SYSTEM Demo
  (* Version 1.0, 2020-01-11, Duc Do Tran *)
  APPLICATION SystemWithoutContract
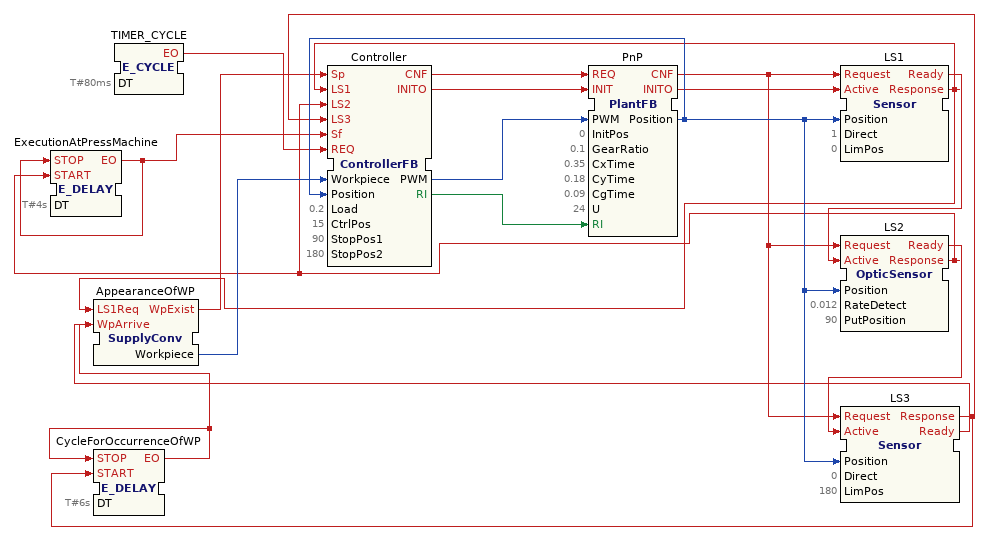
    FBS
      LS2 : OpticSensor(RateDetect := 0.012, PutPosition := 90);
      PnP : PlantFB(InitPos := 0, GearRatio := 0.1, CxTime := 0.35, CyTime := 0.18, CgTime := 0.09, U := 24);
      LS1 : Sensor(Direct := 1, LimPos := 0);
      LS3 : Sensor(Direct := 0, LimPos := 180);
      Controller : ControllerFB(Load := 0.2, CtrlPos := 15, StopPos1 := 90, StopPos2 := 180);
      AppearanceOfWP : SupplyConv;
      ExecutionAtPressMachine : E_DELAY(DT := T#4s);
      CycleForOccurrenceOfWP : E_DELAY(DT := T#6s);
      TIMER_CYCLE : E_CYCLE(DT := T#80ms);
    END_FBS
    EVENT_CONNECTIONS
      PnP.CNF TO LS1.Request;
      PnP.CNF TO LS2.Request;
      PnP.CNF TO LS3.Request;
      PnP.INITO TO LS1.Active;
      LS1.Ready TO LS2.Active;
      LS2.Ready TO LS3.Active;
      Controller.CNF TO PnP.REQ;
      Controller.INITO TO PnP.INIT;
      AppearanceOfWP.WpExist TO Controller.Sp;
      LS1.Response TO AppearanceOfWP.LS1Req;
      LS1.Response TO Controller.LS1;
      LS2.Response TO Controller.LS2;
      LS3.Response TO Controller.LS3;
      ExecutionAtPressMachine.EO TO Controller.Sf;
      ExecutionAtPressMachine.EO TO ExecutionAtPressMachine.STOP;
      CycleForOccurrenceOfWP.EO TO AppearanceOfWP.WpArrive;
      CycleForOccurrenceOfWP.EO TO CycleForOccurrenceOfWP.STOP;
      LS3.Response TO CycleForOccurrenceOfWP.START;
      LS3.Ready TO AppearanceOfWP.WpArrive;
      LS2.Response TO ExecutionAtPressMachine.START;
      TIMER_CYCLE.EO TO Controller.REQ;
    END_CONNECTIONS
    DATA_CONNECTIONS
      PnP.Position TO LS3.Position;
      PnP.Position TO LS2.Position;
      PnP.Position TO LS1.Position;
      Controller.PWM TO PnP.PWM;
      AppearanceOfWP.Workpiece TO Controller.Workpiece;
      PnP.Position TO Controller.Position;
    END_CONNECTIONS
    ADAPTER_CONNECTIONS
      Controller.RI TO PnP.RI;
    END_CONNECTIONS
  END_APPLICATION
  APPLICATION SystemApplyTimingContracts
    FBS
      LS2 : OpticSensor(RateDetect := 0.012, PutPosition := 90);
      ExecutionAtPressMachine : E_DELAY(DT := T#4000ms);
      SplitFirstOccurOfLS1 : SplitInitEv;
      TIMER_CYCLE : E_DELAY(DT := T#20ms);
      LS1ToLS2 : TCFB(QI := 1, GetTime := 0, SetTimeOut := 20.3, Specification := Reaction::q->e(i|=[3.5,4.8]s));
      LS2ToSf : TCFB(QI := 1, GetTime := 0, SetTimeOut := 20.3, Specification := Age::q->e(i|=[3.9,4.4]s));
      SfToLS3 : TCFB(QI := 1, GetTime := 0, SetTimeOut := 20.3, Specification := Reaction::q->e(i|=[4.1,4.6]s));
      LS3ToLS1 : TCFB(QI := 1, GetTime := 0, SetTimeOut := 20.3, Specification := Reaction::q->e(i|=[6.2,6.5]s));
      AppearanceOfWP : SupplyConv;
      PickAndPlaceRobot : PlantFB(InitPos := 0, GearRatio := 0.1, CxTime := 0.35, CyTime := 0.18, CgTime := 0.09, U := 24);
      CycleForOccurrenceOfWP : E_DELAY(DT := T#6000ms);
      LS1 : Sensor(Direct := 1, LimPos := 0);
      LS3 : Sensor(Direct := 0, LimPos := 180);
      Controller : ControllerFB(Load := 0.2, CtrlPos := 15, StopPos1 := 90, StopPos2 := 180);
      EnableCheck : EnableCheck(QIi := 1);
      OnOffLS1 : E_SWITCH(G := 1);
      OnOffLS2 : E_SWITCH(G := 1);
      OnOffLS3 : E_SWITCH(G := 1);
      OnOffFeedingSystem : E_SWITCH(G := 1);
      OnOffPressMachine : E_SWITCH(G := 1);
    END_FBS
    EVENT_CONNECTIONS
      LS2ToSf.Satisfied TO Controller.Sf;
      TIMER_CYCLE.EO TO TIMER_CYCLE.STOP;
      Controller.INITO TO PickAndPlaceRobot.INIT;
      LS2ToSf.INITO TO SfToLS3.INIT;
      SplitFirstOccurOfLS1.CNF TO AppearanceOfWP.LS1Req;
      EnableCheck.Satisfied TO Controller.LS1;
      ExecutionAtPressMachine.EO TO ExecutionAtPressMachine.STOP;
      LS2.Ready TO LS3.Active;
      SfToLS3.INITO TO LS3ToLS1.INIT;
      EnableCheck.Violated TO LS1ToLS2.ReqEvent;
      LS2ToSf.Satisfied TO SfToLS3.ReqEvent;
      CycleForOccurrenceOfWP.EO TO AppearanceOfWP.WpArrive;
      LS3ToLS1.CNF TO TIMER_CYCLE.START;
      EnableCheck.Satisfied TO LS1ToLS2.ReqEvent;
      LS2ToSf.CNF TO SfToLS3.REQ;
      SfToLS3.Satisfied TO Controller.LS3;
      LS2ToSf.Violated TO SfToLS3.ReqEvent;
      PickAndPlaceRobot.INITO TO TIMER_CYCLE.START;
      LS1ToLS2.Violated TO LS2ToSf.ReqEvent;
      SfToLS3.Violated TO LS3ToLS1.ReqEvent;
      TIMER_CYCLE.EO TO LS1ToLS2.REQ;
      LS3ToLS1.Violated TO EnableCheck.REQ;
      LS1ToLS2.Satisfied TO LS2ToSf.ReqEvent;
      LS3ToLS1.CNF TO Controller.REQ;
      LS1ToLS2.Satisfied TO Controller.LS2;
      LS3ToLS1.INITO TO LS1.Active;
      LS3.Response TO SfToLS3.RspEvent;
      LS1.Ready TO LS2.Active;
      LS3.Ready TO AppearanceOfWP.WpArrive;
      ExecutionAtPressMachine.EO TO LS2ToSf.RspEvent;
      LS1ToLS2.INITO TO LS2ToSf.INIT;
      SfToLS3.CNF TO LS3ToLS1.REQ;
      SplitFirstOccurOfLS1.NextTimes TO LS3ToLS1.RspEvent;
      AppearanceOfWP.WpExist TO Controller.Sp;
      LS3ToLS1.Satisfied TO EnableCheck.REQ;
      SfToLS3.Satisfied TO LS3ToLS1.ReqEvent;
      SplitFirstOccurOfLS1.FirstTime TO EnableCheck.REQ;
      LS2.Response TO LS1ToLS2.RspEvent;
      LS3ToLS1.INITO TO Controller.INIT;
      CycleForOccurrenceOfWP.EO TO CycleForOccurrenceOfWP.STOP;
      Controller.CNF TO PickAndPlaceRobot.REQ;
      LS1ToLS2.CNF TO LS2ToSf.REQ;
      LS1.Response TO SplitFirstOccurOfLS1.REQ;
      PickAndPlaceRobot.CNF TO OnOffLS3.EI;
      OnOffLS3.EO1 TO LS3.Request;
      PickAndPlaceRobot.CNF TO OnOffLS2.EI;
      OnOffLS2.EO1 TO LS2.Request;
      PickAndPlaceRobot.CNF TO OnOffLS1.EI;
      OnOffLS1.EO1 TO LS1.Request;
      LS3.Response TO OnOffFeedingSystem.EI;
      OnOffFeedingSystem.EO1 TO CycleForOccurrenceOfWP.START;
      LS1ToLS2.Satisfied TO OnOffPressMachine.EI;
      OnOffPressMachine.EO1 TO ExecutionAtPressMachine.START;
    END_CONNECTIONS
    DATA_CONNECTIONS
      PickAndPlaceRobot.Position TO LS3.Position;
      LS1ToLS2.QO TO LS2ToSf.QI;
      PickAndPlaceRobot.Position TO LS1.Position;
      Controller.PWM TO PickAndPlaceRobot.PWM;
      EnableCheck.OUT TO LS1ToLS2.QI;
      PickAndPlaceRobot.Position TO LS2.Position;
      LS2ToSf.QO TO SfToLS3.QI;
      PickAndPlaceRobot.Position TO Controller.Position;
      LS3ToLS1.QO TO EnableCheck.QIt;
      SfToLS3.QO TO LS3ToLS1.QI;
      AppearanceOfWP.Workpiece TO Controller.Workpiece;
    END_CONNECTIONS
    ADAPTER_CONNECTIONS
      Controller.RI TO PickAndPlaceRobot.RI;
    END_CONNECTIONS
  END_APPLICATION
  DEVICE FORTE_PC : FORTE_PC(MGR_ID := "localhost:61499")
    {SET_ATTRIBUTE(Profile, HOLOBLOC)} (* device profile *)
    RESOURCE CPU1 : EMB_RES
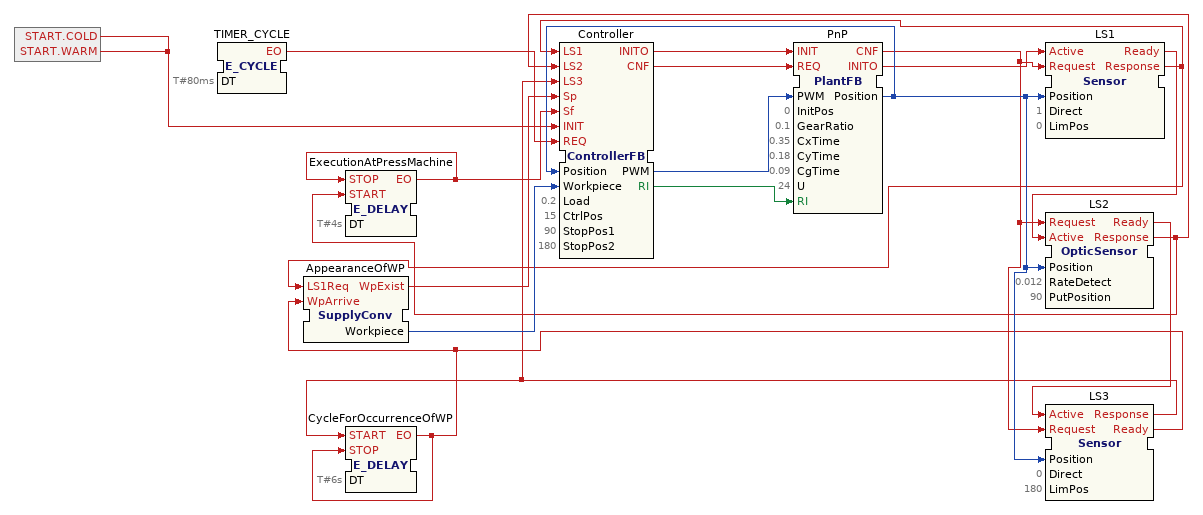
      FBS
        LS2 : OpticSensor(RateDetect := 0.012, PutPosition := 90);
        PnP : PlantFB(InitPos := 0, GearRatio := 0.1, CxTime := 0.35, CyTime := 0.18, CgTime := 0.09, U := 24);
        LS1 : Sensor(Direct := 1, LimPos := 0);
        LS3 : Sensor(Direct := 0, LimPos := 180);
        Controller : ControllerFB(Load := 0.2, CtrlPos := 15, StopPos1 := 90, StopPos2 := 180);
        AppearanceOfWP : SupplyConv;
        ExecutionAtPressMachine : E_DELAY(DT := T#4s);
        CycleForOccurrenceOfWP : E_DELAY(DT := T#6s);
        TIMER_CYCLE : E_CYCLE(DT := T#80ms);
      END_FBS
      EVENT_CONNECTIONS
        PnP.CNF TO LS2.Request;
        PnP.INITO TO LS1.Active;
        PnP.CNF TO LS1.Request;
        LS1.Ready TO LS2.Active;
        LS2.Ready TO LS3.Active;
        PnP.CNF TO LS3.Request;
        LS1.Response TO Controller.LS1;
        LS2.Response TO Controller.LS2;
        LS3.Response TO Controller.LS3;
        Controller.INITO TO PnP.INIT;
        Controller.CNF TO PnP.REQ;
        LS1.Response TO AppearanceOfWP.LS1Req;
        AppearanceOfWP.WpExist TO Controller.Sp;
        ExecutionAtPressMachine.EO TO ExecutionAtPressMachine.STOP;
        ExecutionAtPressMachine.EO TO Controller.Sf;
        LS3.Response TO CycleForOccurrenceOfWP.START;
        CycleForOccurrenceOfWP.EO TO CycleForOccurrenceOfWP.STOP;
        CycleForOccurrenceOfWP.EO TO AppearanceOfWP.WpArrive;
        LS3.Ready TO AppearanceOfWP.WpArrive;
        LS2.Response TO ExecutionAtPressMachine.START;
        START.COLD TO Controller.INIT;
        START.WARM TO Controller.INIT;
        TIMER_CYCLE.EO TO Controller.REQ;
      END_CONNECTIONS
      DATA_CONNECTIONS
        PnP.Position TO LS2.Position;
        PnP.Position TO LS1.Position;
        PnP.Position TO LS3.Position;
        PnP.Position TO Controller.Position;
        Controller.PWM TO PnP.PWM;
        AppearanceOfWP.Workpiece TO Controller.Workpiece;
      END_CONNECTIONS
      ADAPTER_CONNECTIONS
        Controller.RI TO PnP.RI;
      END_CONNECTIONS
    END_RESOURCE
    RESOURCE CPU2 : EMB_RES
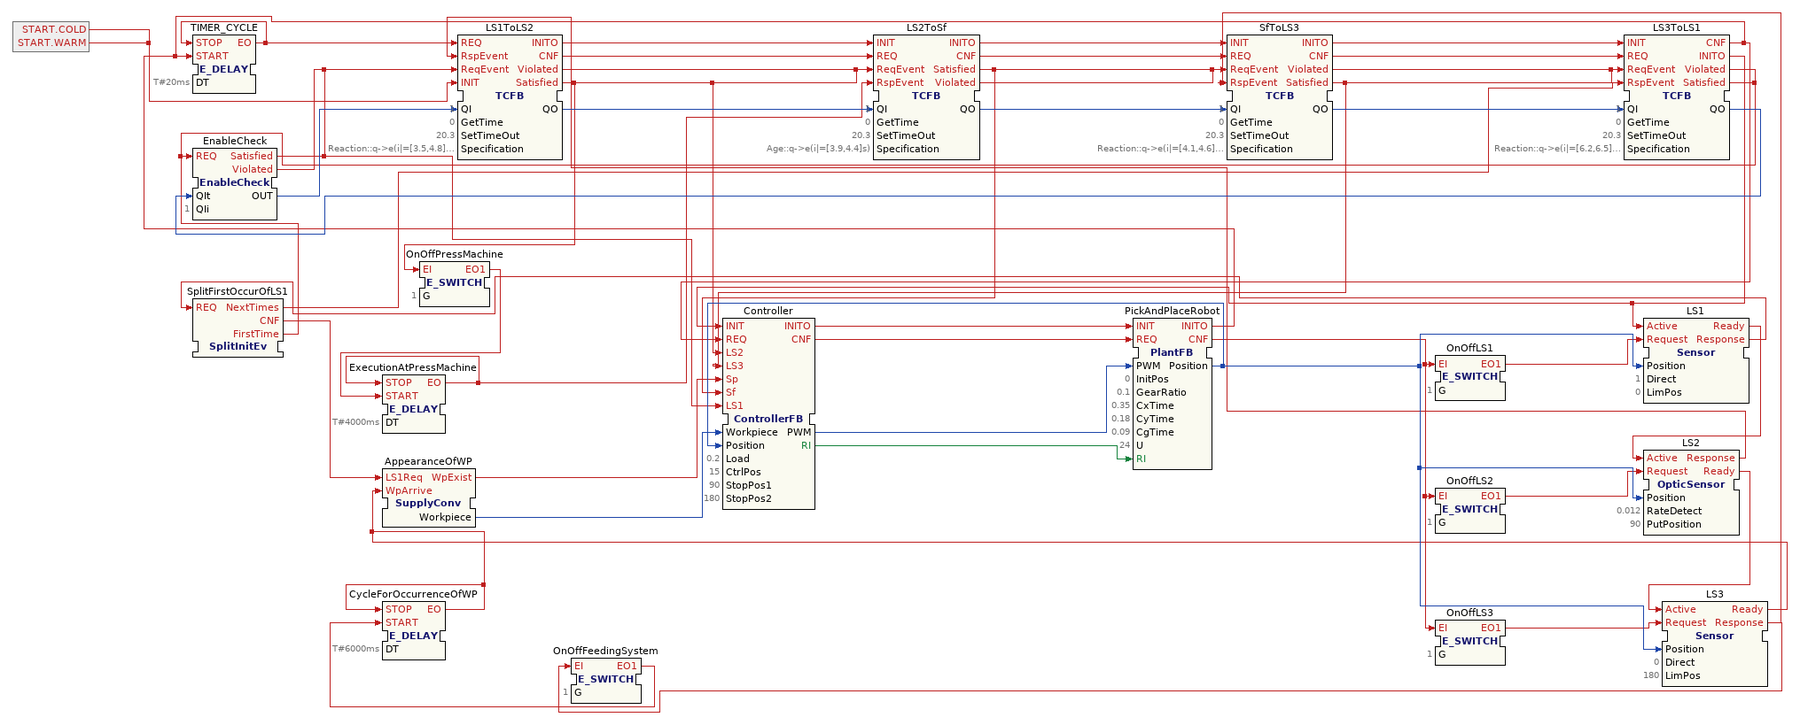
      FBS
        LS2 : OpticSensor(RateDetect := 0.012, PutPosition := 90);
        ExecutionAtPressMachine : E_DELAY(DT := T#4000ms);
        SplitFirstOccurOfLS1 : SplitInitEv;
        TIMER_CYCLE : E_DELAY(DT := T#20ms);
        LS1ToLS2 : TCFB(QI := 1, GetTime := 0, SetTimeOut := 20.3, Specification := Reaction::q->e(i|=[3.5,4.8]s));
        LS2ToSf : TCFB(QI := 1, GetTime := 0, SetTimeOut := 20.3, Specification := Age::q->e(i|=[3.9,4.4]s));
        SfToLS3 : TCFB(QI := 1, GetTime := 0, SetTimeOut := 20.3, Specification := Reaction::q->e(i|=[4.1,4.6]s));
        LS3ToLS1 : TCFB(QI := 1, GetTime := 0, SetTimeOut := 20.3, Specification := Reaction::q->e(i|=[6.2,6.5]s));
        AppearanceOfWP : SupplyConv;
        PickAndPlaceRobot : PlantFB(InitPos := 0, GearRatio := 0.1, CxTime := 0.35, CyTime := 0.18, CgTime := 0.09, U := 24);
        CycleForOccurrenceOfWP : E_DELAY(DT := T#6000ms);
        LS1 : Sensor(Direct := 1, LimPos := 0);
        LS3 : Sensor(Direct := 0, LimPos := 180);
        Controller : ControllerFB(Load := 0.2, CtrlPos := 15, StopPos1 := 90, StopPos2 := 180);
        EnableCheck : EnableCheck(QIi := 1);
        OnOffPressMachine : E_SWITCH(G := 1);
        OnOffFeedingSystem : E_SWITCH(G := 1);
        OnOffLS2 : E_SWITCH(G := 1);
        OnOffLS1 : E_SWITCH(G := 1);
        OnOffLS3 : E_SWITCH(G := 1);
      END_FBS
      EVENT_CONNECTIONS
        ExecutionAtPressMachine.EO TO ExecutionAtPressMachine.STOP;
        TIMER_CYCLE.EO TO TIMER_CYCLE.STOP;
        TIMER_CYCLE.EO TO LS1ToLS2.REQ;
        LS2.Response TO LS1ToLS2.RspEvent;
        LS1ToLS2.INITO TO LS2ToSf.INIT;
        LS1ToLS2.CNF TO LS2ToSf.REQ;
        LS1ToLS2.Violated TO LS2ToSf.ReqEvent;
        LS1ToLS2.Satisfied TO LS2ToSf.ReqEvent;
        ExecutionAtPressMachine.EO TO LS2ToSf.RspEvent;
        LS2ToSf.INITO TO SfToLS3.INIT;
        LS2ToSf.CNF TO SfToLS3.REQ;
        LS2ToSf.Satisfied TO SfToLS3.ReqEvent;
        LS2ToSf.Violated TO SfToLS3.ReqEvent;
        SfToLS3.INITO TO LS3ToLS1.INIT;
        SfToLS3.CNF TO LS3ToLS1.REQ;
        SfToLS3.Violated TO LS3ToLS1.ReqEvent;
        SfToLS3.Satisfied TO LS3ToLS1.ReqEvent;
        SplitFirstOccurOfLS1.NextTimes TO LS3ToLS1.RspEvent;
        LS3ToLS1.CNF TO TIMER_CYCLE.START;
        SplitFirstOccurOfLS1.CNF TO AppearanceOfWP.LS1Req;
        PickAndPlaceRobot.INITO TO TIMER_CYCLE.START;
        CycleForOccurrenceOfWP.EO TO CycleForOccurrenceOfWP.STOP;
        CycleForOccurrenceOfWP.EO TO AppearanceOfWP.WpArrive;
        LS3ToLS1.INITO TO LS1.Active;
        LS1.Ready TO LS2.Active;
        LS2.Ready TO LS3.Active;
        LS3.Ready TO AppearanceOfWP.WpArrive;
        LS3.Response TO SfToLS3.RspEvent;
        LS3ToLS1.INITO TO Controller.INIT;
        LS3ToLS1.CNF TO Controller.REQ;
        LS1ToLS2.Satisfied TO Controller.LS2;
        SfToLS3.Satisfied TO Controller.LS3;
        AppearanceOfWP.WpExist TO Controller.Sp;
        LS2ToSf.Satisfied TO Controller.Sf;
        Controller.INITO TO PickAndPlaceRobot.INIT;
        Controller.CNF TO PickAndPlaceRobot.REQ;
        LS3ToLS1.Violated TO EnableCheck.REQ;
        LS3ToLS1.Satisfied TO EnableCheck.REQ;
        SplitFirstOccurOfLS1.FirstTime TO EnableCheck.REQ;
        EnableCheck.Satisfied TO Controller.LS1;
        EnableCheck.Satisfied TO LS1ToLS2.ReqEvent;
        EnableCheck.Violated TO LS1ToLS2.ReqEvent;
        START.COLD TO LS1ToLS2.INIT;
        START.WARM TO LS1ToLS2.INIT;
        LS1.Response TO SplitFirstOccurOfLS1.REQ;
        LS1ToLS2.Satisfied TO OnOffPressMachine.EI;
        OnOffPressMachine.EO1 TO ExecutionAtPressMachine.START;
        LS3.Response TO OnOffFeedingSystem.EI;
        OnOffFeedingSystem.EO1 TO CycleForOccurrenceOfWP.START;
        PickAndPlaceRobot.CNF TO OnOffLS2.EI;
        OnOffLS2.EO1 TO LS2.Request;
        PickAndPlaceRobot.CNF TO OnOffLS1.EI;
        OnOffLS1.EO1 TO LS1.Request;
        PickAndPlaceRobot.CNF TO OnOffLS3.EI;
        OnOffLS3.EO1 TO LS3.Request;
      END_CONNECTIONS
      DATA_CONNECTIONS
        LS1ToLS2.QO TO LS2ToSf.QI;
        LS2ToSf.QO TO SfToLS3.QI;
        SfToLS3.QO TO LS3ToLS1.QI;
        PickAndPlaceRobot.Position TO LS2.Position;
        PickAndPlaceRobot.Position TO LS1.Position;
        PickAndPlaceRobot.Position TO LS3.Position;
        AppearanceOfWP.Workpiece TO Controller.Workpiece;
        PickAndPlaceRobot.Position TO Controller.Position;
        Controller.PWM TO PickAndPlaceRobot.PWM;
        LS3ToLS1.QO TO EnableCheck.QIt;
        EnableCheck.OUT TO LS1ToLS2.QI;
      END_CONNECTIONS
      ADAPTER_CONNECTIONS
        Controller.RI TO PickAndPlaceRobot.RI;
      END_CONNECTIONS
    END_RESOURCE
  END_DEVICE
  MAPPINGS
    SystemWithoutContract.LS2 ON FORTE_PC.CPU1.LS2;
    SystemWithoutContract.PnP ON FORTE_PC.CPU1.PnP;
    SystemWithoutContract.LS1 ON FORTE_PC.CPU1.LS1;
    SystemWithoutContract.LS3 ON FORTE_PC.CPU1.LS3;
    SystemWithoutContract.Controller ON FORTE_PC.CPU1.Controller;
    SystemWithoutContract.AppearanceOfWP ON FORTE_PC.CPU1.AppearanceOfWP;
    SystemWithoutContract.ExecutionAtPressMachine ON FORTE_PC.CPU1.ExecutionAtPressMachine;
    SystemWithoutContract.CycleForOccurrenceOfWP ON FORTE_PC.CPU1.CycleForOccurrenceOfWP;
    SystemWithoutContract.TIMER_CYCLE ON FORTE_PC.CPU1.TIMER_CYCLE;
    SystemApplyTimingContracts.LS2 ON FORTE_PC.CPU2.LS2;
    SystemApplyTimingContracts.ExecutionAtPressMachine ON FORTE_PC.CPU2.ExecutionAtPressMachine;
    SystemApplyTimingContracts.SplitFirstOccurOfLS1 ON FORTE_PC.CPU2.SplitFirstOccurOfLS1;
    SystemApplyTimingContracts.TIMER_CYCLE ON FORTE_PC.CPU2.TIMER_CYCLE;
    SystemApplyTimingContracts.LS1ToLS2 ON FORTE_PC.CPU2.LS1ToLS2;
    SystemApplyTimingContracts.LS2ToSf ON FORTE_PC.CPU2.LS2ToSf;
    SystemApplyTimingContracts.SfToLS3 ON FORTE_PC.CPU2.SfToLS3;
    SystemApplyTimingContracts.LS3ToLS1 ON FORTE_PC.CPU2.LS3ToLS1;
    SystemApplyTimingContracts.AppearanceOfWP ON FORTE_PC.CPU2.AppearanceOfWP;
    SystemApplyTimingContracts.PickAndPlaceRobot ON FORTE_PC.CPU2.PickAndPlaceRobot;
    SystemApplyTimingContracts.CycleForOccurrenceOfWP ON FORTE_PC.CPU2.CycleForOccurrenceOfWP;
    SystemApplyTimingContracts.LS1 ON FORTE_PC.CPU2.LS1;
    SystemApplyTimingContracts.LS3 ON FORTE_PC.CPU2.LS3;
    SystemApplyTimingContracts.Controller ON FORTE_PC.CPU2.Controller;
    SystemApplyTimingContracts.EnableCheck ON FORTE_PC.CPU2.EnableCheck;
    SystemApplyTimingContracts.OnOffPressMachine ON FORTE_PC.CPU2.OnOffPressMachine;
    SystemApplyTimingContracts.OnOffFeedingSystem ON FORTE_PC.CPU2.OnOffFeedingSystem;
    SystemApplyTimingContracts.OnOffLS2 ON FORTE_PC.CPU2.OnOffLS2;
    SystemApplyTimingContracts.OnOffLS1 ON FORTE_PC.CPU2.OnOffLS1;
    SystemApplyTimingContracts.OnOffLS3 ON FORTE_PC.CPU2.OnOffLS3;
  END_MAPPINGS
  SEGMENTS
    Ethernet : Ethernet;
  END_SEGMENTS
  LINKS
    FORTE_PC => Ethernet;
  END_LINKS
END_SYSTEM
